PROGRAM PRG_08_ProductionStatistics
VAR
	PartsPerMinInstant					: PartsPerMinInstant2;
	PartsPerMin							: GenericState;
	PartsPerMinPublishMqtt				: PublishJsonMqtt;
	OkPartsPerMinHistorical				: PartsPerMinHistorical;
END_VAR

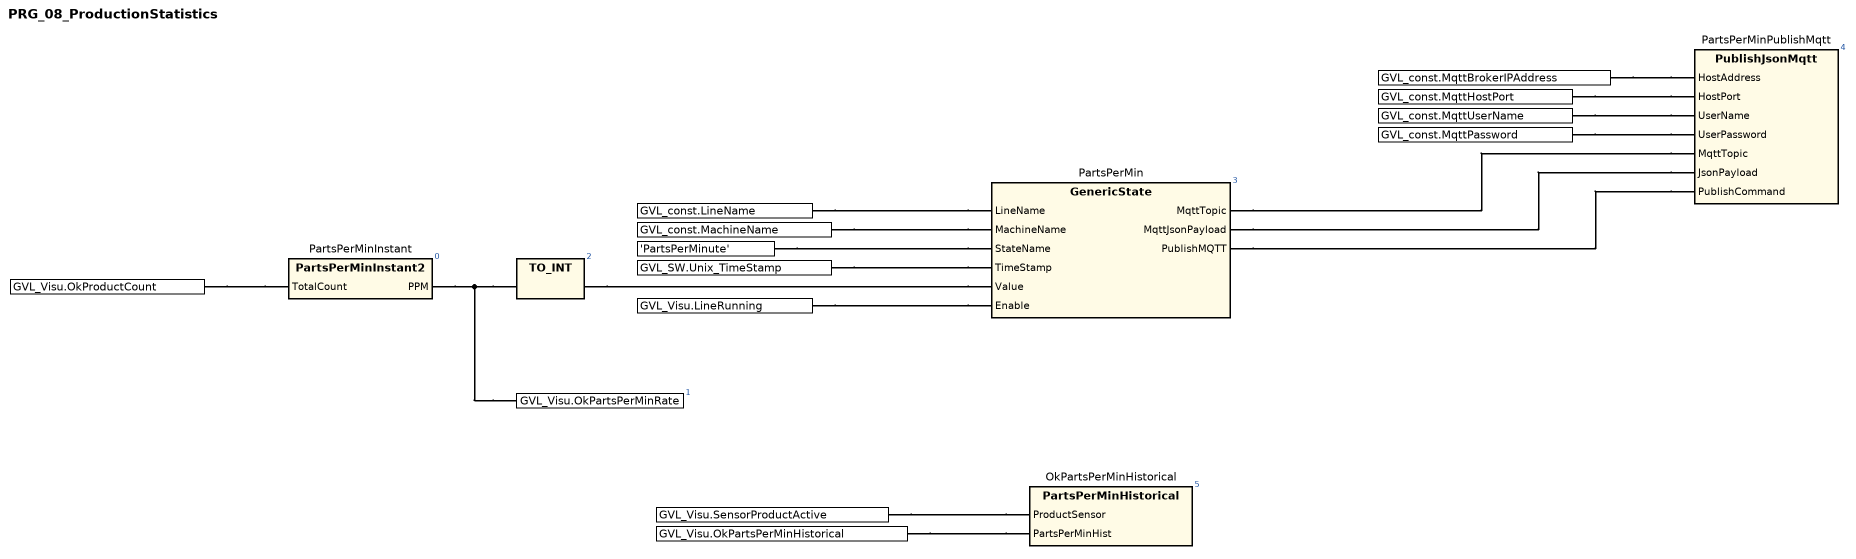
PartsPerMinInstant(TotalCount := GVL_Visu.OkProductCount); // PartsPerMinInstant2
GVL_Visu.OkPartsPerMinRate := PartsPerMinInstant.PPM;
PartsPerMin(
    LineName := GVL_const.LineName,
    MachineName := GVL_const.MachineName,
    StateName := 'PartsPerMinute',
    TimeStamp := GVL_SW.Unix_TimeStamp,
    Value := TO_INT(PartsPerMinInstant.PPM),
    Enable := GVL_Visu.LineRunning); // GenericState
PartsPerMinPublishMqtt(
    HostAddress := GVL_const.MqttBrokerIPAddress,
    HostPort := GVL_const.MqttHostPort,
    UserName := GVL_const.MqttUserName,
    UserPassword := GVL_const.MqttPassword,
    MqttTopic := PartsPerMin.MqttTopic,
    JsonPayload := PartsPerMin.MqttJsonPayload,
    PublishCommand := PartsPerMin.PublishMQTT); // PublishJsonMqtt
OkPartsPerMinHistorical(ProductSensor := GVL_Visu.SensorProductActive, PartsPerMinHist := GVL_Visu.OkPartsPerMinHistorical); // PartsPerMinHistorical

END_PROGRAM

(* stored: Version 1.1.0.1, ProductVersion 3.1.4024.15
   POU PRG_08_ProductionStatistics: Id {fd94bcd0-a2f7-44a7-96a3-f0f108da018e}, SpecialFunc None *)
